Staubli VAL3: deleteItem.pgx

program deleteItem(bool& x_bResult)
  local string l_sSwap
  local num l_nResult
  local string l_sMessage
  local string l_sMessage2
  local bool l_bYes
  local string l_sButton[2]
  local InstrItem l_iSwap
begin
  //
  // delete a Trajectory
  //
  x_bResult=false
  // check
  if sEvent!=""
    l_iSwap.sType=saveData:sTrajTypeUsing
    l_iSwap.sData=sEvent
    call prog:findItem(l_iSwap,l_nResult,false)
    if l_nResult==0
      //delete it
      call language:message(l_sMessage,81)
      call language:getYesNo(l_sButton)
      // ask the yes_no question
      call use:yes_no(l_sMessage+"#"+saveData:sTrajTypeUsing+" "+sEvent,l_sButton,l_bYes)
      x_bResult=l_bYes
    endIf
  endIf
end
